// SIMATIC S7-200 SMART project (STEP 7-Micro/WIN SMART), CPU ST20

SYMBOL_TABLE System Symbols
Always_On        SM0.0    // Always ON
END_SYMBOL_TABLE

ORGANIZATION_BLOCK MAIN:OB1
TITLE=Program Comments
BEGIN
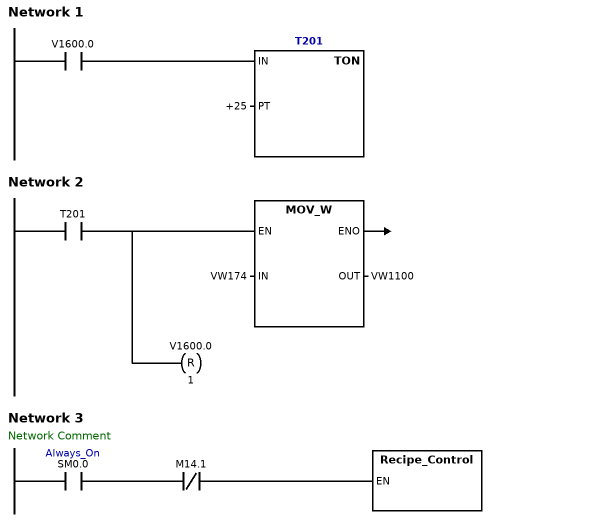
Network 1
LD     V1600.0
TON    T201, +25
Network 2
LD     T201
MOVW   VW174, VW1100
R      V1600.0, 1
Network 3
// Network Comment
LD     Always_On:SM0.0
AN     M14.1
CALL   Recipe_Control:SBR0
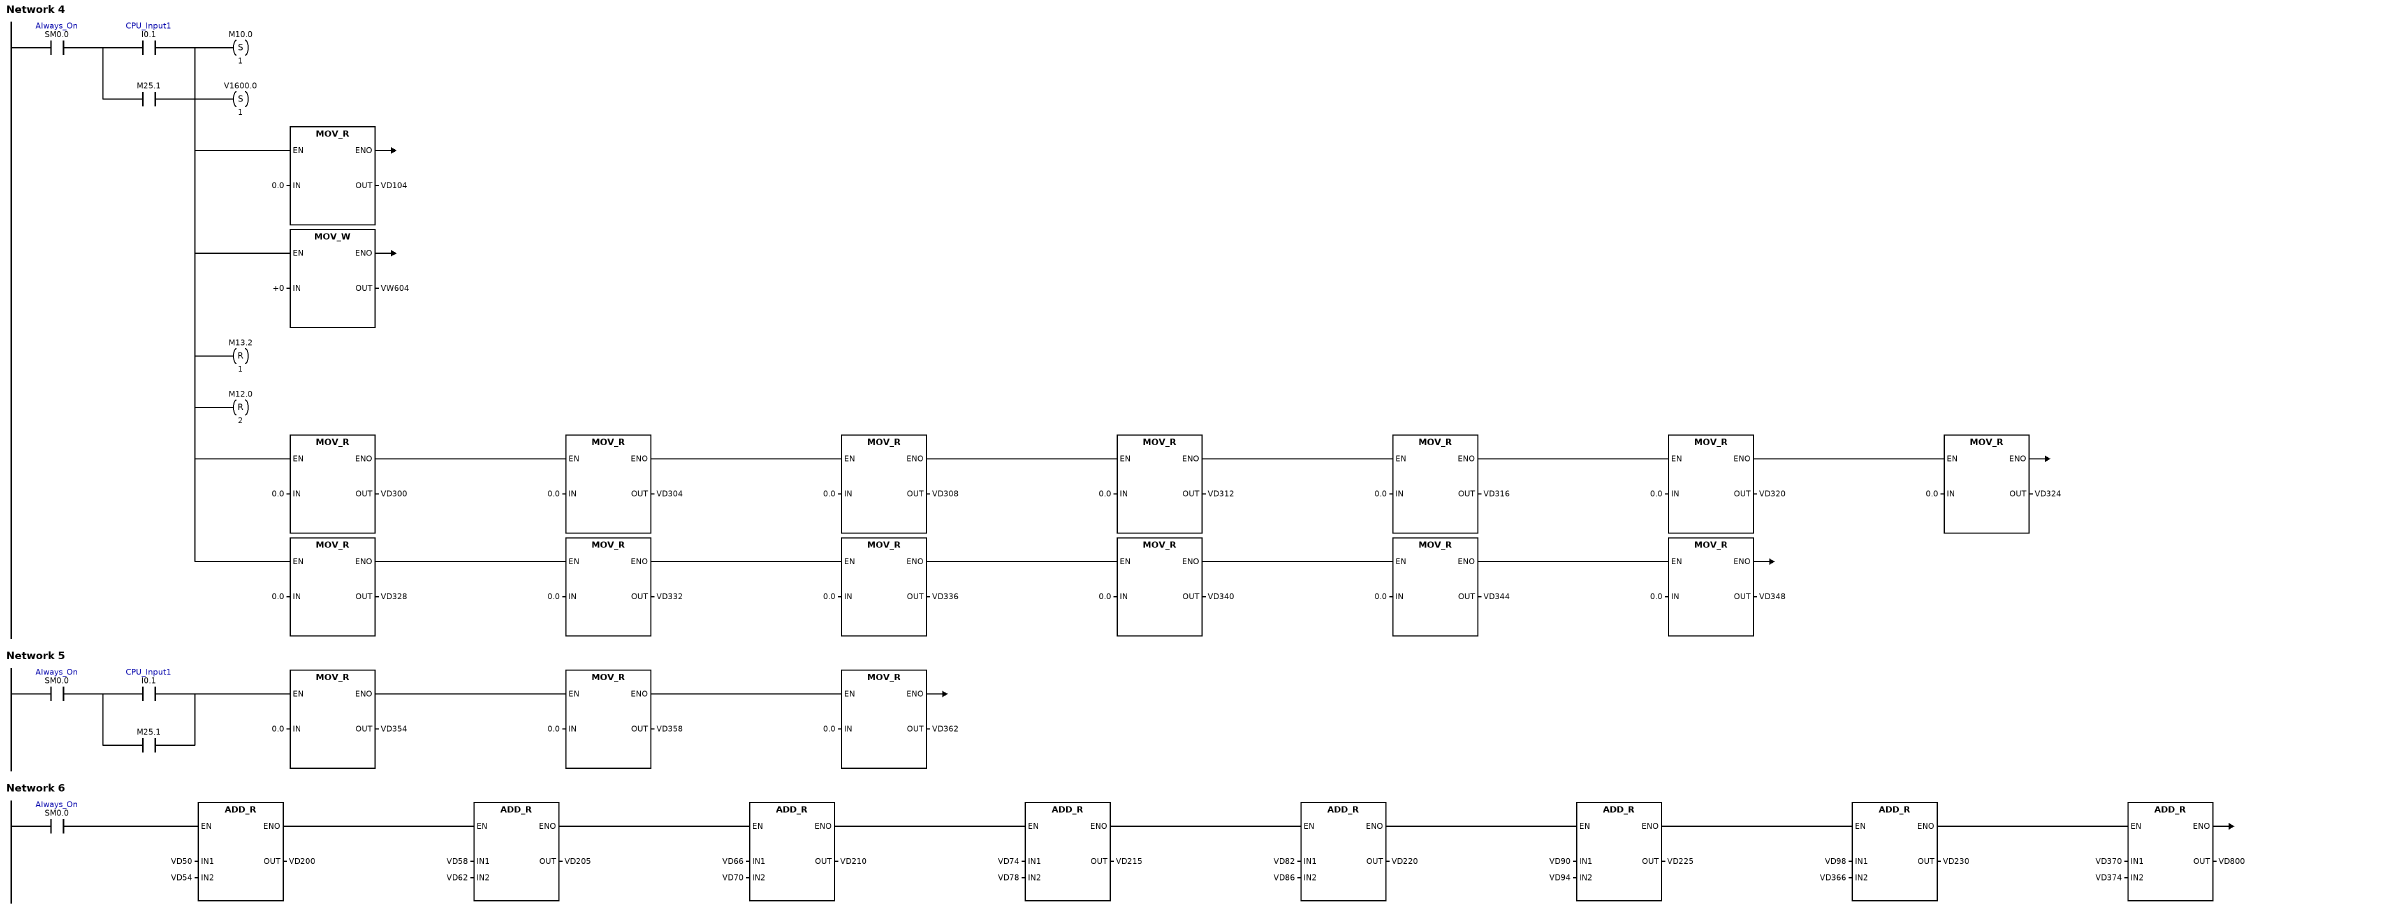
Network 4
LD     Always_On:SM0.0
LD     CPU_Input1:I0.1
O      M25.1
ALD
LPS
S      M10.0, 1
S      V1600.0, 1
MOVR   0.0, VD104
MOVW   +0, VW604
R      M13.2, 1
R      M12.0, 2
MOVR   0.0, VD300
AENO
MOVR   0.0, VD304
AENO
MOVR   0.0, VD308
AENO
MOVR   0.0, VD312
AENO
MOVR   0.0, VD316
AENO
MOVR   0.0, VD320
AENO
MOVR   0.0, VD324
LPP
MOVR   0.0, VD328
AENO
MOVR   0.0, VD332
AENO
MOVR   0.0, VD336
AENO
MOVR   0.0, VD340
AENO
MOVR   0.0, VD344
AENO
MOVR   0.0, VD348
Network 5
LD     Always_On:SM0.0
LD     CPU_Input1:I0.1
O      M25.1
ALD
MOVR   0.0, VD354
AENO
MOVR   0.0, VD358
AENO
MOVR   0.0, VD362
Network 6
LD     Always_On:SM0.0
MOVR   VD50, VD200
AENO
+R     VD54, VD200
AENO
MOVR   VD58, VD205
AENO
+R     VD62, VD205
AENO
MOVR   VD66, VD210
AENO
+R     VD70, VD210
AENO
MOVR   VD74, VD215
AENO
+R     VD78, VD215
AENO
MOVR   VD82, VD220
AENO
+R     VD86, VD220
AENO
MOVR   VD90, VD225
AENO
+R     VD94, VD225
AENO
MOVR   VD98, VD230
AENO
+R     VD366, VD230
AENO
MOVR   VD370, VD800
+R     VD374, VD800
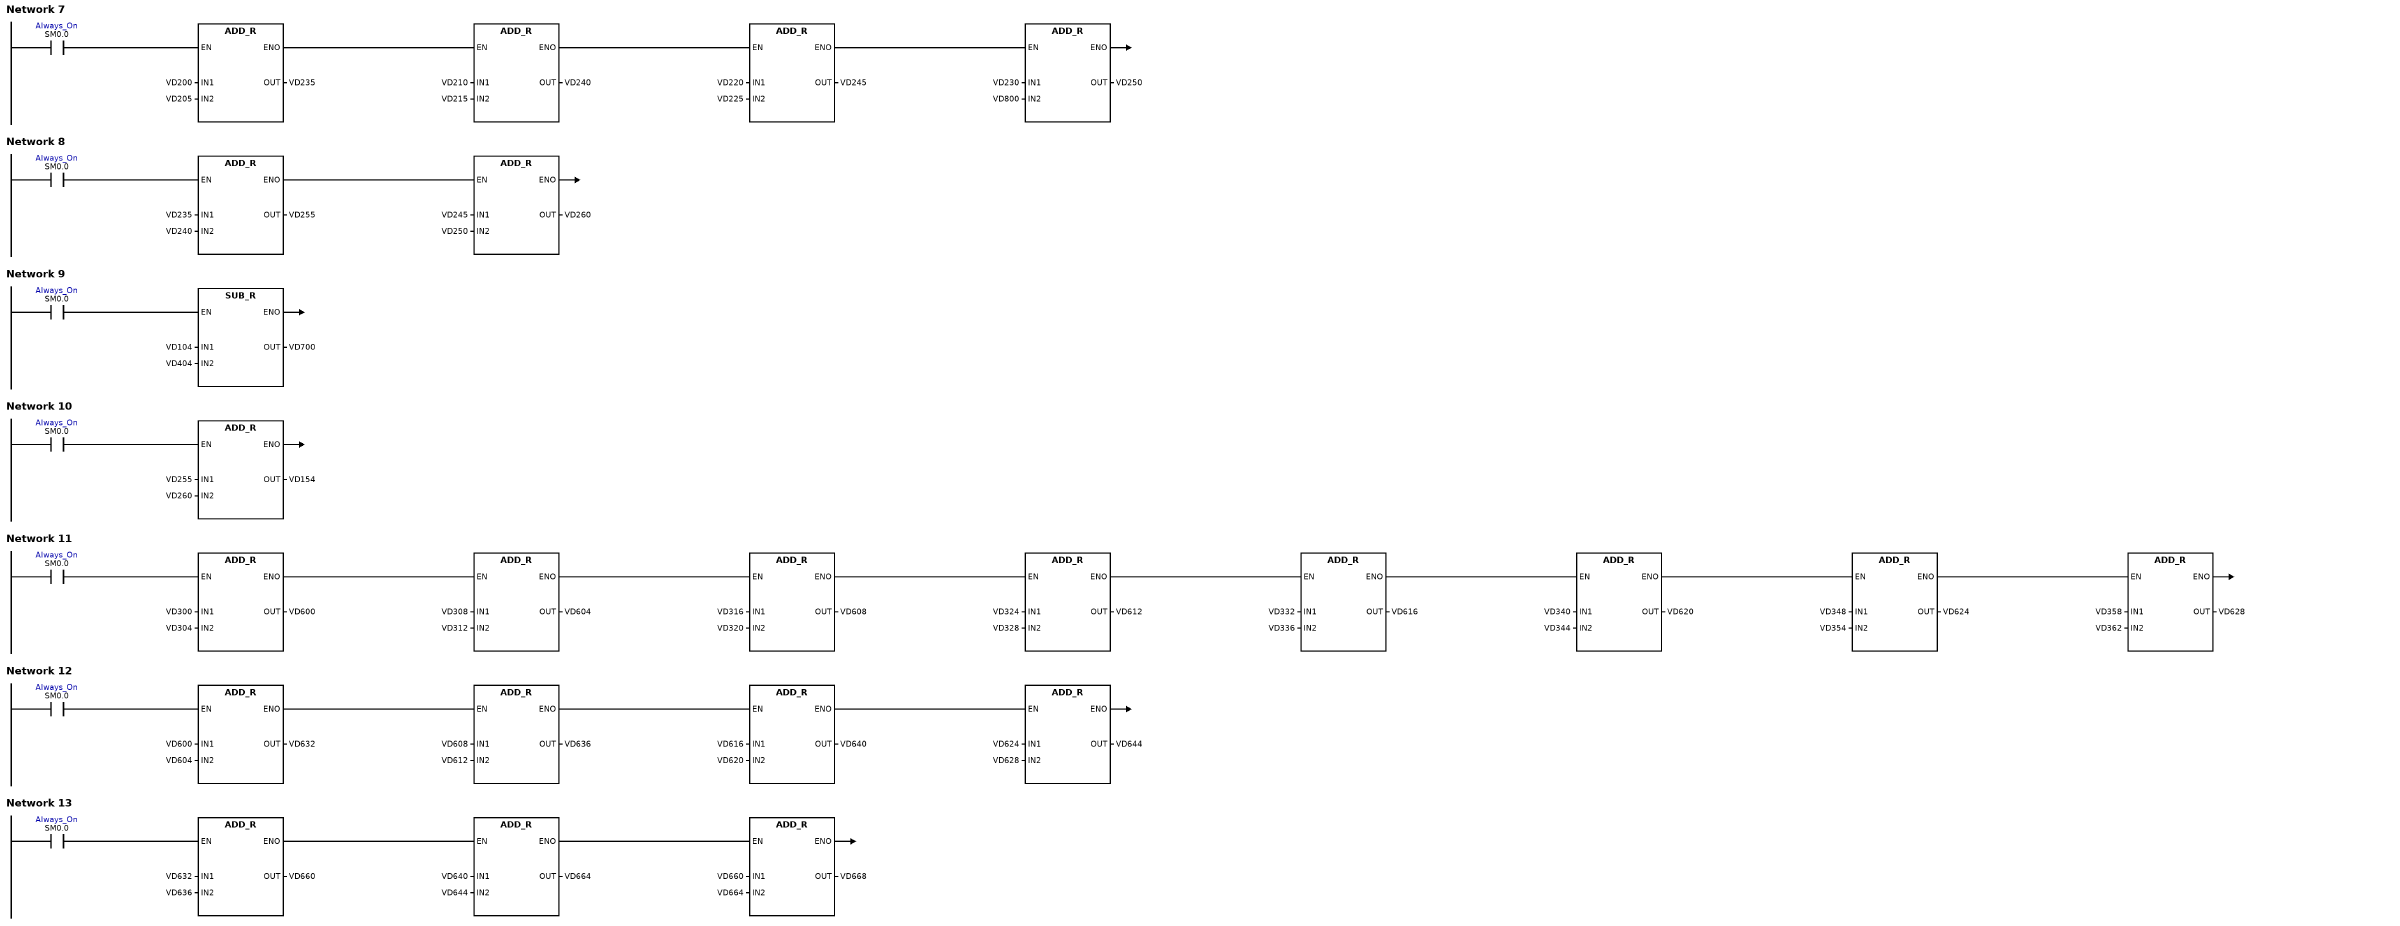
Network 7
LD     Always_On:SM0.0
MOVR   VD200, VD235
AENO
+R     VD205, VD235
AENO
MOVR   VD210, VD240
AENO
+R     VD215, VD240
AENO
MOVR   VD220, VD245
AENO
+R     VD225, VD245
AENO
MOVR   VD230, VD250
+R     VD800, VD250
Network 8
LD     Always_On:SM0.0
MOVR   VD235, VD255
AENO
+R     VD240, VD255
AENO
MOVR   VD245, VD260
+R     VD250, VD260
Network 9
LD     Always_On:SM0.0
MOVR   VD104, VD700
-R     VD404, VD700
Network 10
LD     Always_On:SM0.0
MOVR   VD255, VD154
+R     VD260, VD154
Network 11
LD     Always_On:SM0.0
MOVR   VD300, VD600
AENO
+R     VD304, VD600
AENO
MOVR   VD308, VD604
AENO
+R     VD312, VD604
AENO
MOVR   VD316, VD608
AENO
+R     VD320, VD608
AENO
MOVR   VD324, VD612
AENO
+R     VD328, VD612
AENO
MOVR   VD332, VD616
AENO
+R     VD336, VD616
AENO
MOVR   VD340, VD620
AENO
+R     VD344, VD620
AENO
MOVR   VD348, VD624
AENO
+R     VD354, VD624
AENO
MOVR   VD358, VD628
+R     VD362, VD628
Network 12
LD     Always_On:SM0.0
MOVR   VD600, VD632
AENO
+R     VD604, VD632
AENO
MOVR   VD608, VD636
AENO
+R     VD612, VD636
AENO
MOVR   VD616, VD640
AENO
+R     VD620, VD640
AENO
MOVR   VD624, VD644
+R     VD628, VD644
Network 13
LD     Always_On:SM0.0
MOVR   VD632, VD660
AENO
+R     VD636, VD660
AENO
MOVR   VD640, VD664
AENO
+R     VD644, VD664
AENO
MOVR   VD660, VD668
+R     VD664, VD668
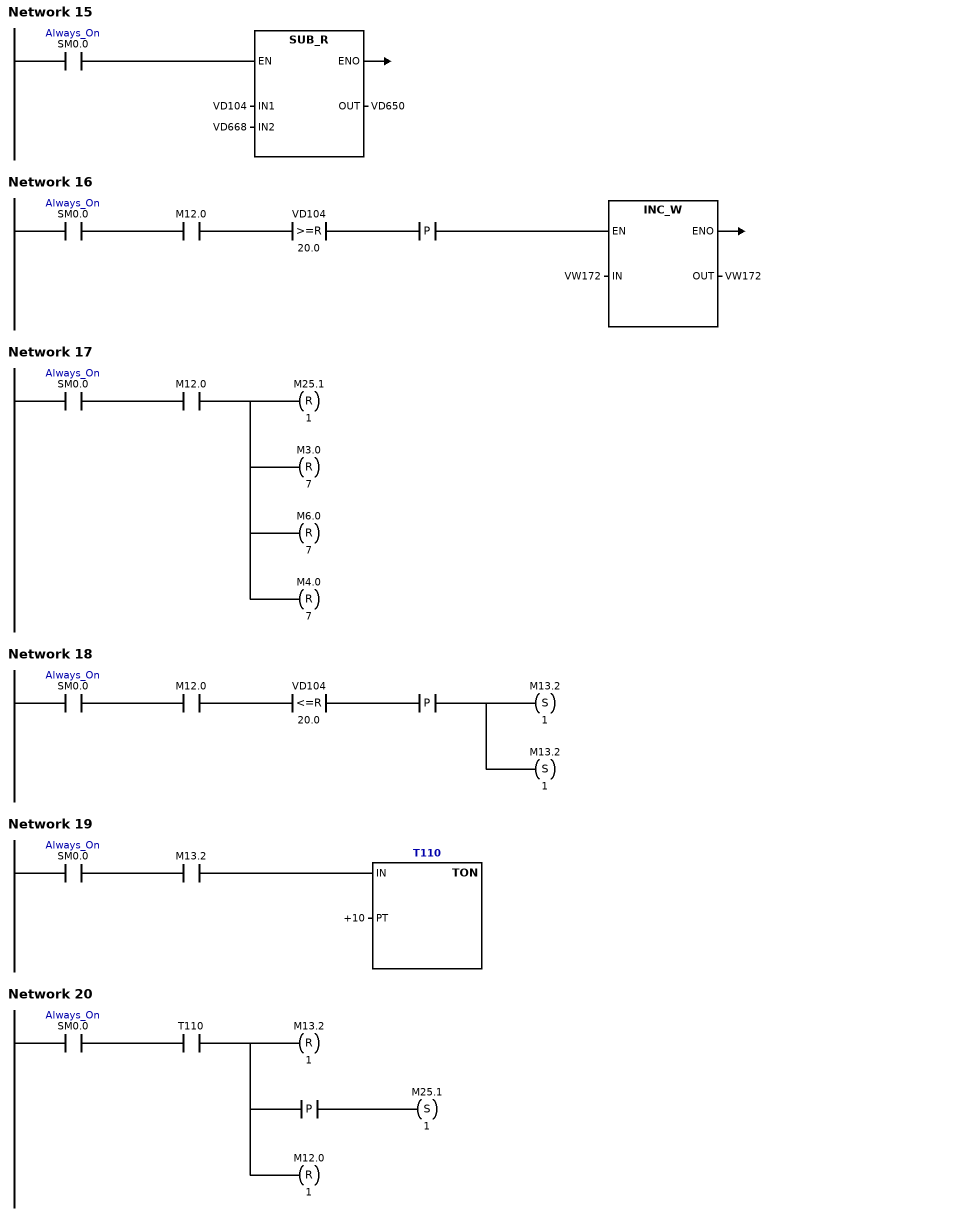
Network 15
LD     Always_On:SM0.0
MOVR   VD104, VD650
-R     VD668, VD650
Network 16
LD     Always_On:SM0.0
A      M12.0
AR>=   VD104, 20.0
EU
INCW   VW172
Network 17
LD     Always_On:SM0.0
A      M12.0
R      M25.1, 1
R      M3.0, 7
R      M6.0, 7
R      M4.0, 7
Network 18
LD     Always_On:SM0.0
A      M12.0
AR<=   VD104, 20.0
EU
S      M13.2, 1
S      M13.2, 1
Network 19
LD     Always_On:SM0.0
A      M13.2
TON    T110, +10
Network 20
LD     Always_On:SM0.0
A      T110
LPS
R      M13.2, 1
EU
S      M25.1, 1
LPP
R      M12.0, 1
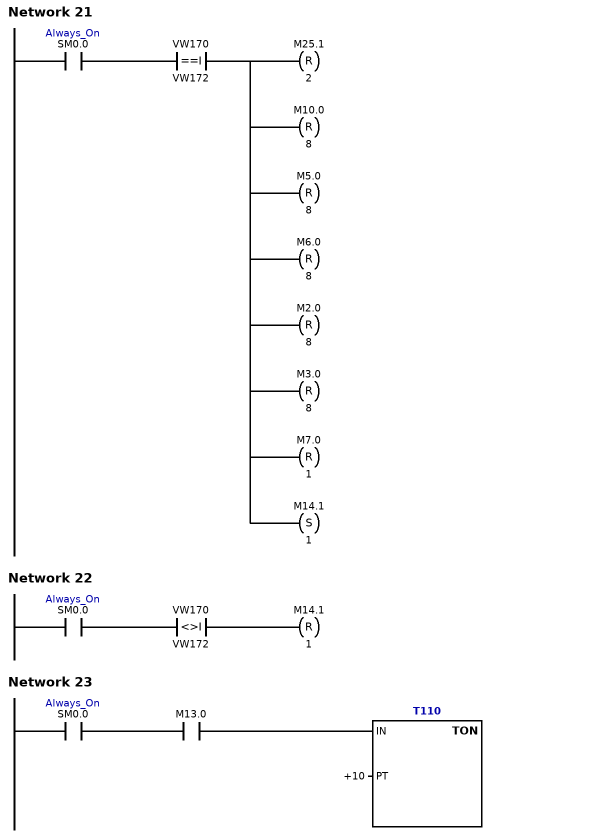
Network 21
LD     Always_On:SM0.0
AW=    VW170, VW172
R      M25.1, 2
R      M10.0, 8
R      M5.0, 8
R      M6.0, 8
R      M2.0, 8
R      M3.0, 8
R      M7.0, 1
S      M14.1, 1
Network 22
LD     Always_On:SM0.0
AW<>   VW170, VW172
R      M14.1, 1
Network 23
LD     Always_On:SM0.0
A      M13.0
TON    T110, +10
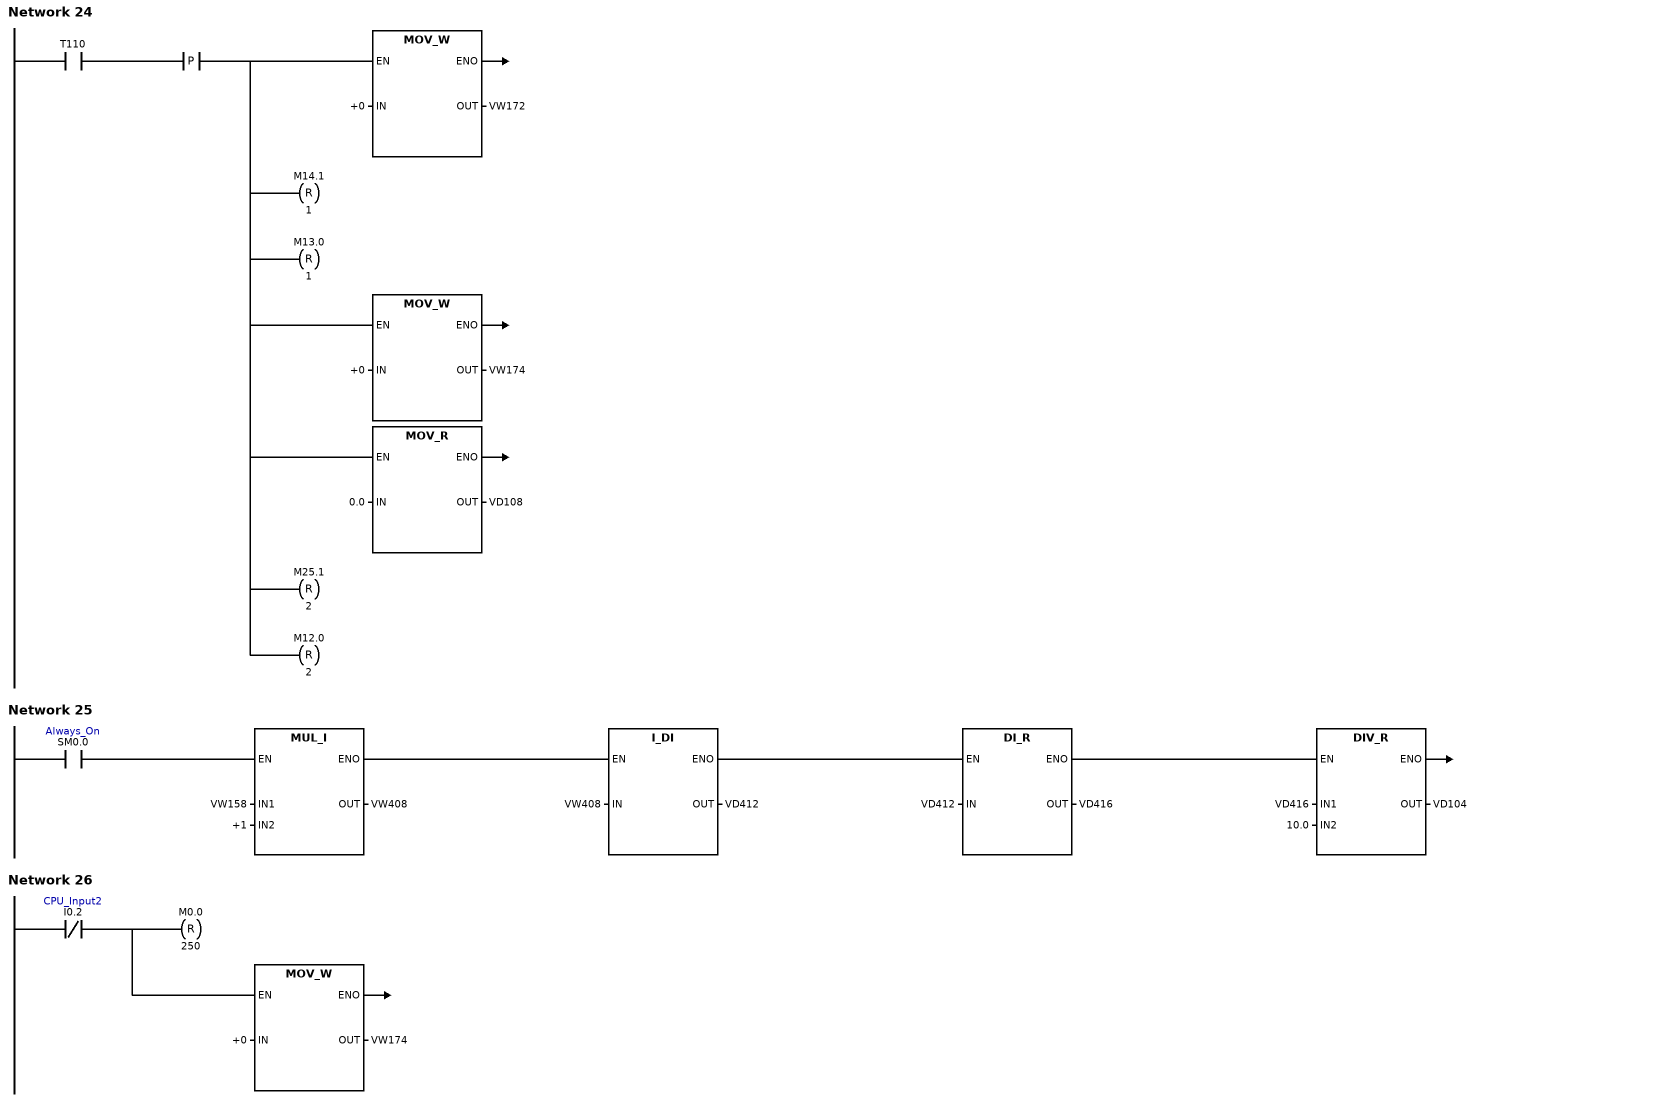
Network 24
LD     T110
EU
MOVW   +0, VW172
R      M14.1, 1
R      M13.0, 1
MOVW   +0, VW174
MOVR   0.0, VD108
R      M25.1, 2
R      M12.0, 2
Network 25
LD     Always_On:SM0.0
MOVW   VW158, VW408
AENO
*I     +1, VW408
AENO
ITD    VW408, VD412
AENO
DTR    VD412, VD416
AENO
MOVR   VD416, VD104
/R     10.0, VD104
Network 26
LDN    CPU_Input2:I0.2
R      M0.0, 250
MOVW   +0, VW174
END_ORGANIZATION_BLOCK

SUBROUTINE_BLOCK Recipe_Control:SBR0
TITLE=Subroutine Comments
BEGIN
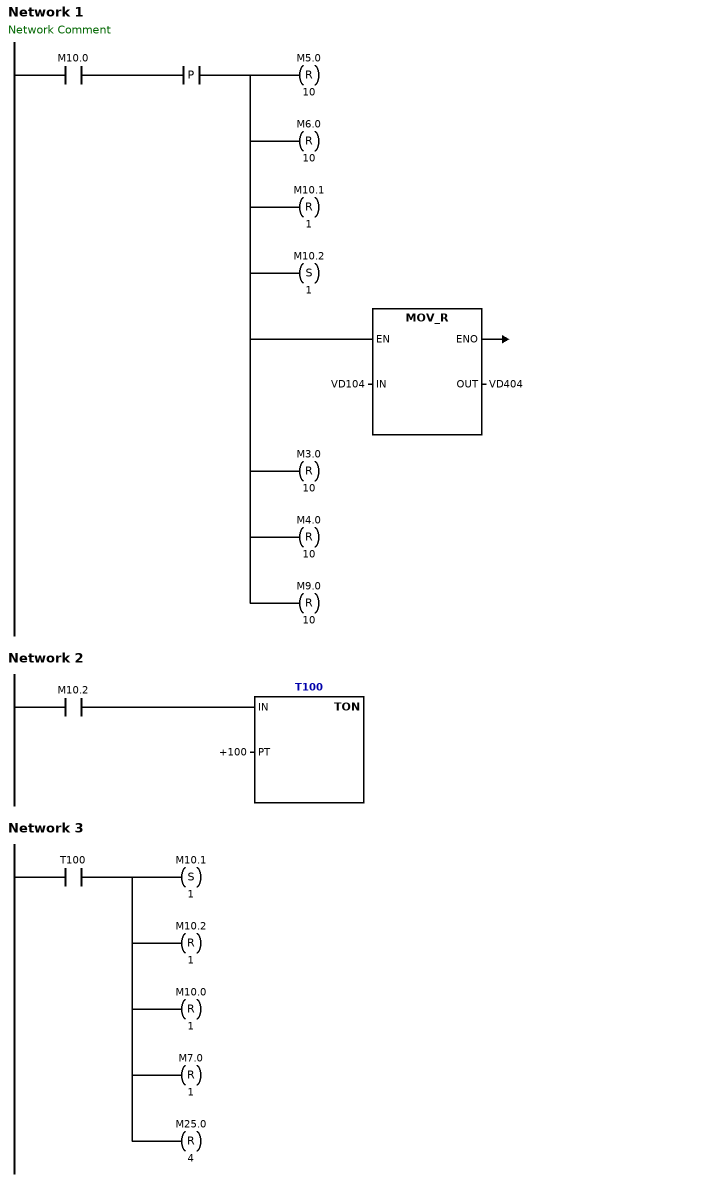
Network 1
// Network Comment
LD     M10.0
EU
R      M5.0, 10
R      M6.0, 10
R      M10.1, 1
S      M10.2, 1
MOVR   VD104, VD404
R      M3.0, 10
R      M4.0, 10
R      M9.0, 10
Network 2
LD     M10.2
TON    T100, +100
Network 3
LD     T100
S      M10.1, 1
R      M10.2, 1
R      M10.0, 1
R      M7.0, 1
R      M25.0, 4
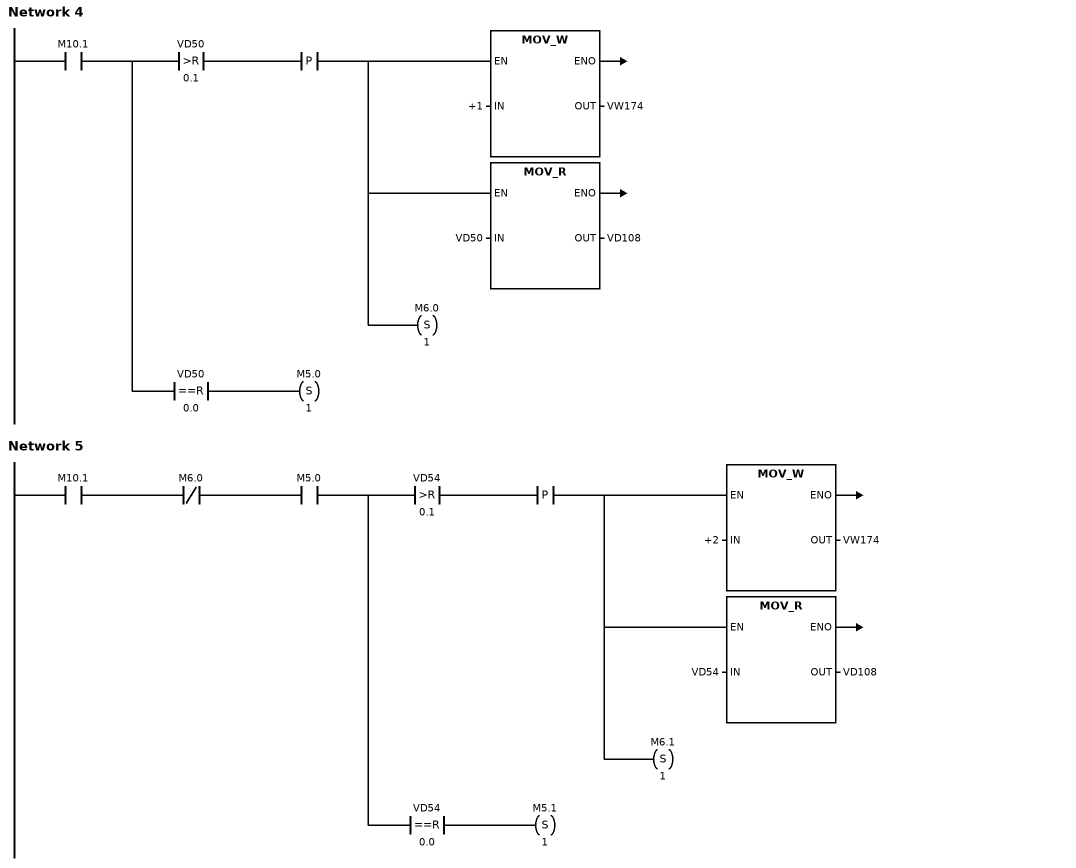
Network 4
LD     M10.1
LPS
AR>    VD50, 0.1
EU
MOVW   +1, VW174
MOVR   VD50, VD108
S      M6.0, 1
LPP
AR=    VD50, 0.0
S      M5.0, 1
Network 5
LD     M10.1
AN     M6.0
A      M5.0
LPS
AR>    VD54, 0.1
EU
MOVW   +2, VW174
MOVR   VD54, VD108
S      M6.1, 1
LPP
AR=    VD54, 0.0
S      M5.1, 1
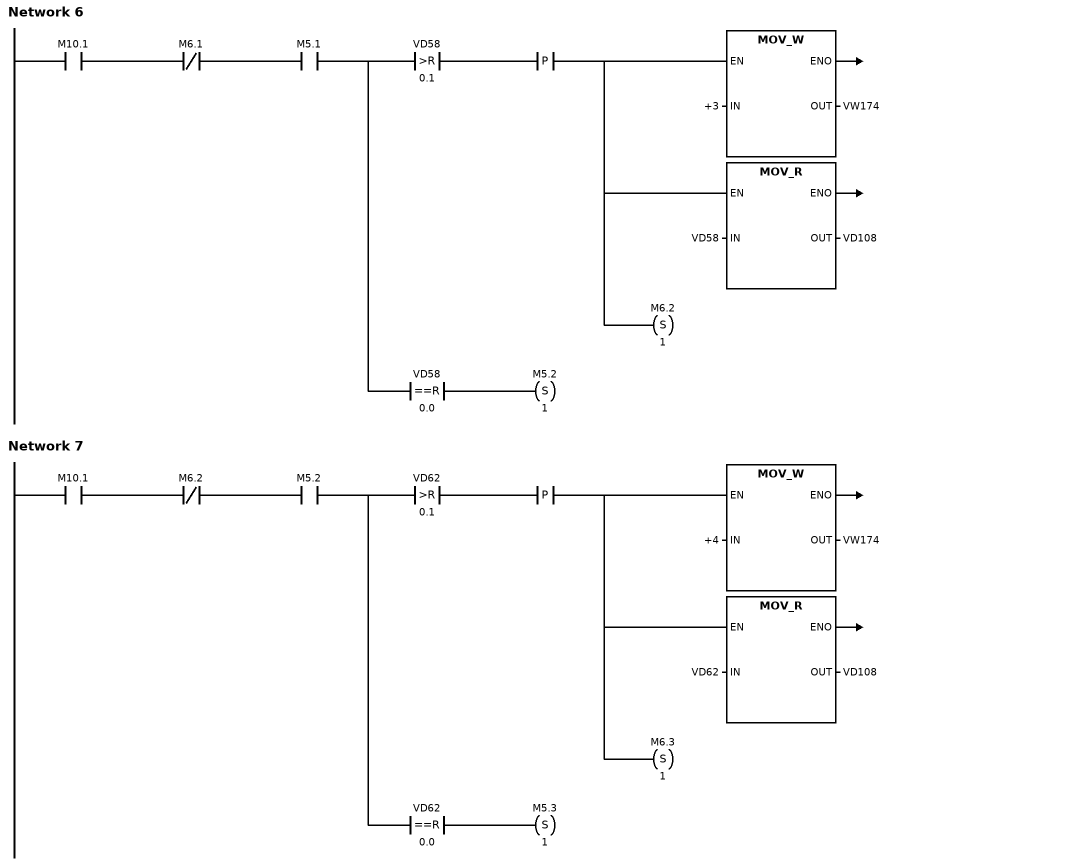
Network 6
LD     M10.1
AN     M6.1
A      M5.1
LPS
AR>    VD58, 0.1
EU
MOVW   +3, VW174
MOVR   VD58, VD108
S      M6.2, 1
LPP
AR=    VD58, 0.0
S      M5.2, 1
Network 7
LD     M10.1
AN     M6.2
A      M5.2
LPS
AR>    VD62, 0.1
EU
MOVW   +4, VW174
MOVR   VD62, VD108
S      M6.3, 1
LPP
AR=    VD62, 0.0
S      M5.3, 1
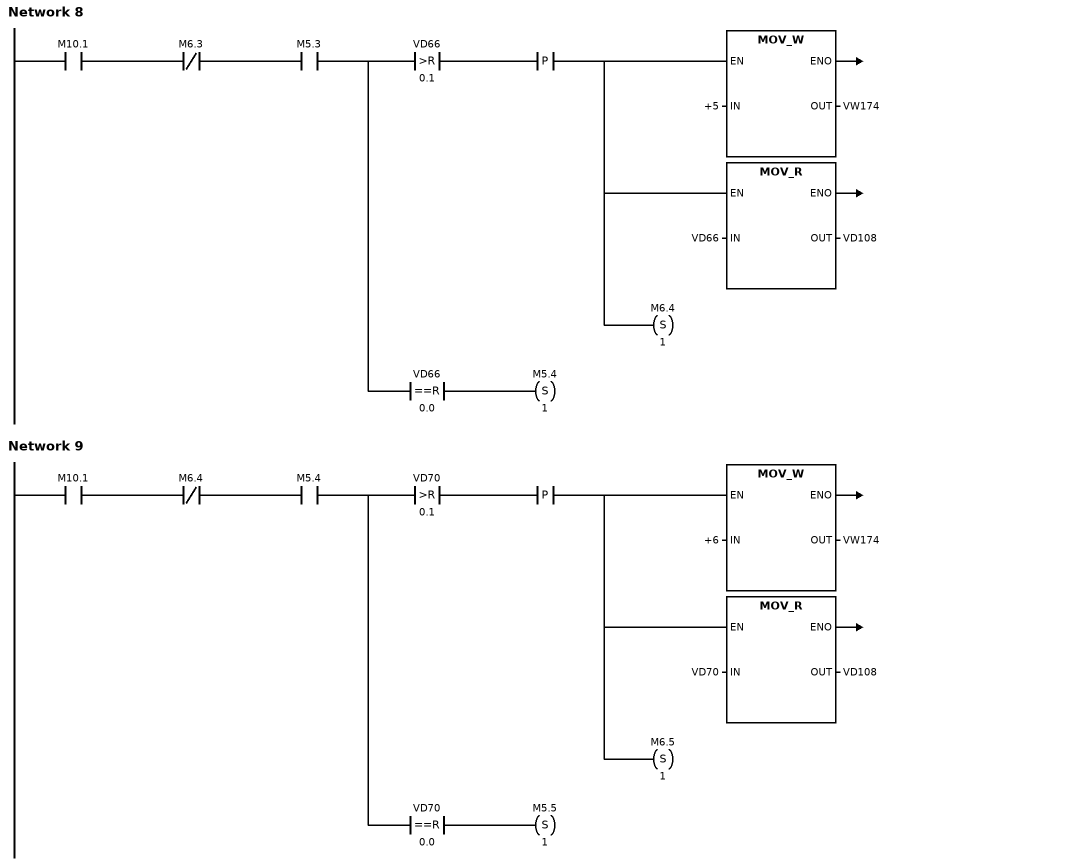
Network 8
LD     M10.1
AN     M6.3
A      M5.3
LPS
AR>    VD66, 0.1
EU
MOVW   +5, VW174
MOVR   VD66, VD108
S      M6.4, 1
LPP
AR=    VD66, 0.0
S      M5.4, 1
Network 9
LD     M10.1
AN     M6.4
A      M5.4
LPS
AR>    VD70, 0.1
EU
MOVW   +6, VW174
MOVR   VD70, VD108
S      M6.5, 1
LPP
AR=    VD70, 0.0
S      M5.5, 1
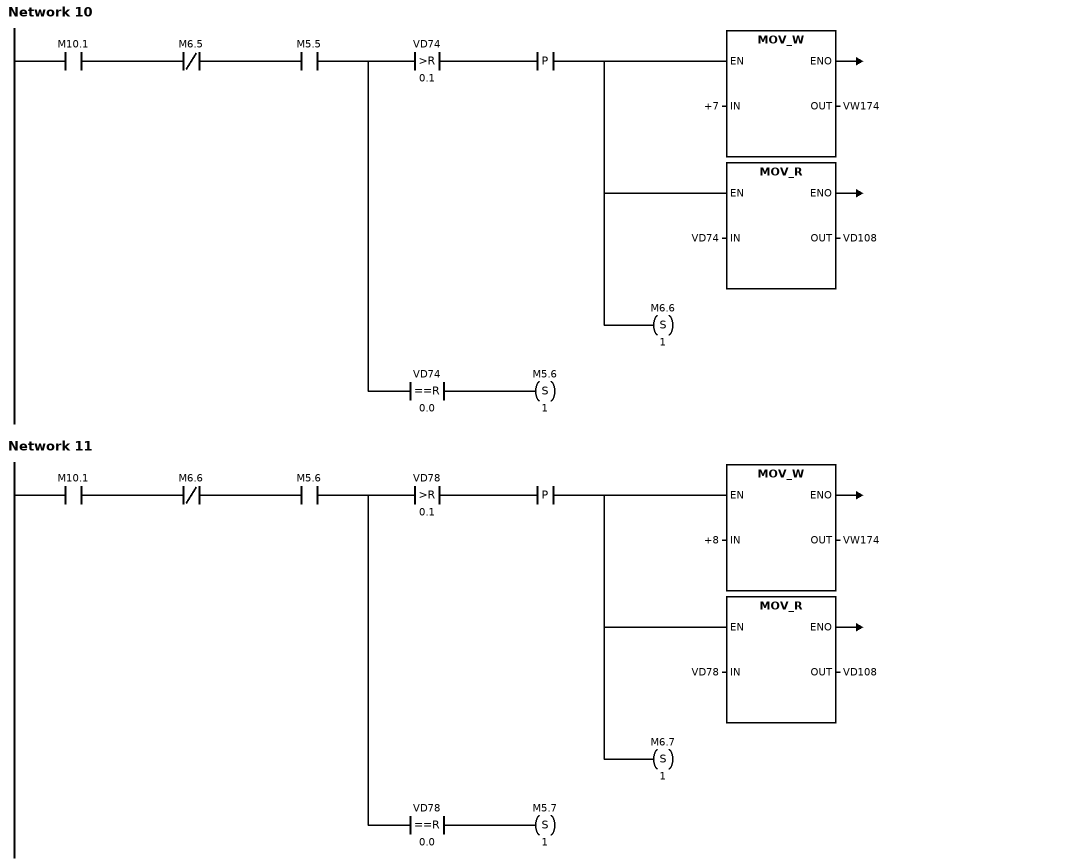
Network 10
LD     M10.1
AN     M6.5
A      M5.5
LPS
AR>    VD74, 0.1
EU
MOVW   +7, VW174
MOVR   VD74, VD108
S      M6.6, 1
LPP
AR=    VD74, 0.0
S      M5.6, 1
Network 11
LD     M10.1
AN     M6.6
A      M5.6
LPS
AR>    VD78, 0.1
EU
MOVW   +8, VW174
MOVR   VD78, VD108
S      M6.7, 1
LPP
AR=    VD78, 0.0
S      M5.7, 1
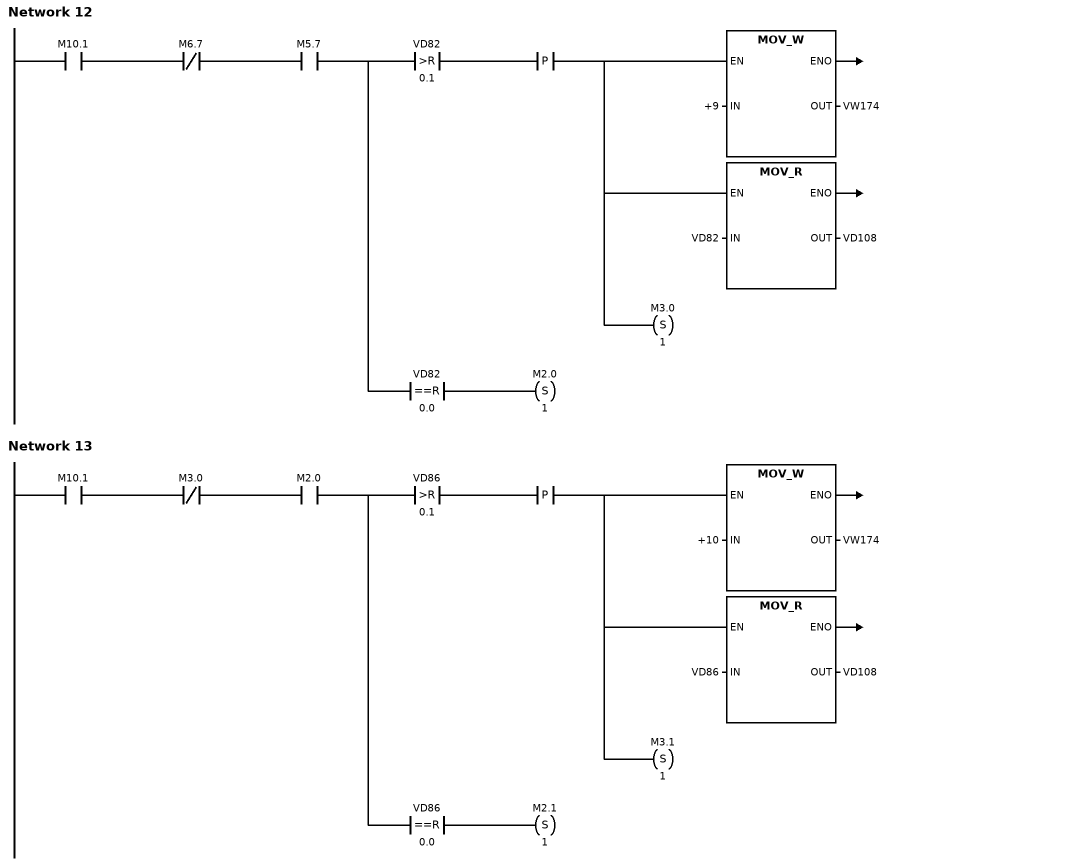
Network 12
LD     M10.1
AN     M6.7
A      M5.7
LPS
AR>    VD82, 0.1
EU
MOVW   +9, VW174
MOVR   VD82, VD108
S      M3.0, 1
LPP
AR=    VD82, 0.0
S      M2.0, 1
Network 13
LD     M10.1
AN     M3.0
A      M2.0
LPS
AR>    VD86, 0.1
EU
MOVW   +10, VW174
MOVR   VD86, VD108
S      M3.1, 1
LPP
AR=    VD86, 0.0
S      M2.1, 1
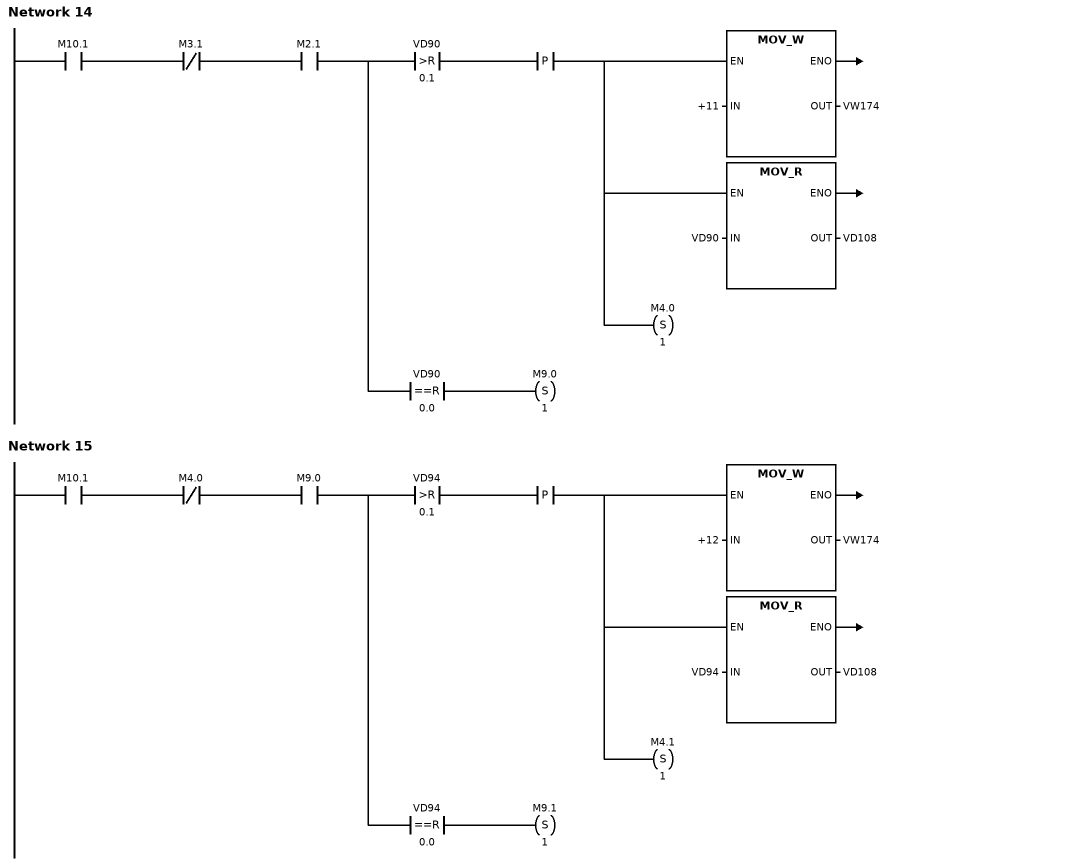
Network 14
LD     M10.1
AN     M3.1
A      M2.1
LPS
AR>    VD90, 0.1
EU
MOVW   +11, VW174
MOVR   VD90, VD108
S      M4.0, 1
LPP
AR=    VD90, 0.0
S      M9.0, 1
Network 15
LD     M10.1
AN     M4.0
A      M9.0
LPS
AR>    VD94, 0.1
EU
MOVW   +12, VW174
MOVR   VD94, VD108
S      M4.1, 1
LPP
AR=    VD94, 0.0
S      M9.1, 1
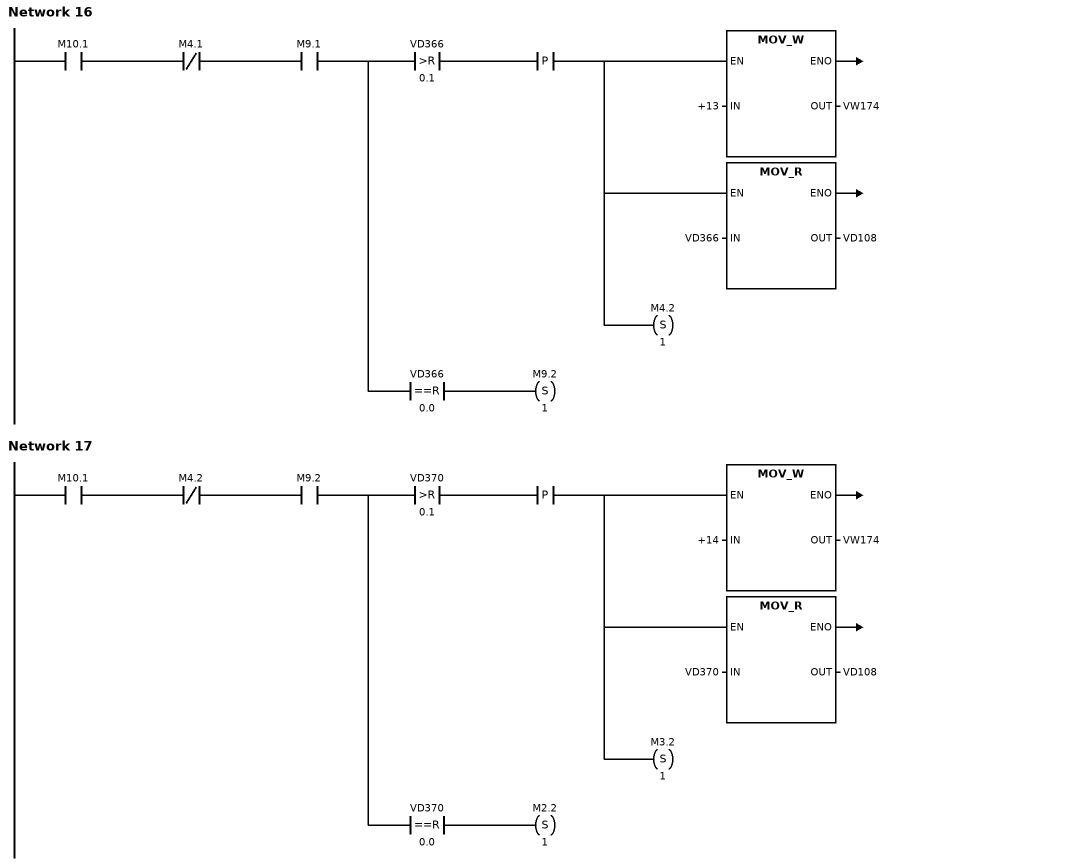
Network 16
LD     M10.1
AN     M4.1
A      M9.1
LPS
AR>    VD366, 0.1
EU
MOVW   +13, VW174
MOVR   VD366, VD108
S      M4.2, 1
LPP
AR=    VD366, 0.0
S      M9.2, 1
Network 17
LD     M10.1
AN     M4.2
A      M9.2
LPS
AR>    VD370, 0.1
EU
MOVW   +14, VW174
MOVR   VD370, VD108
S      M3.2, 1
LPP
AR=    VD370, 0.0
S      M2.2, 1
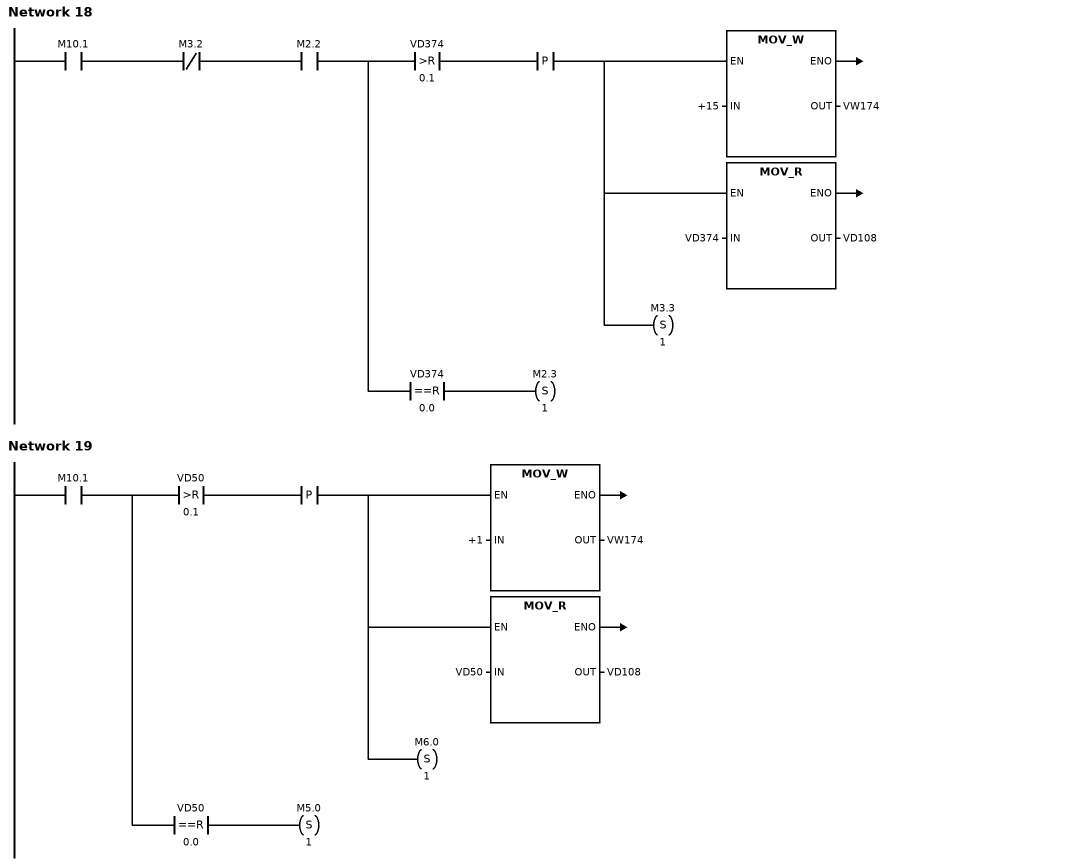
Network 18
LD     M10.1
AN     M3.2
A      M2.2
LPS
AR>    VD374, 0.1
EU
MOVW   +15, VW174
MOVR   VD374, VD108
S      M3.3, 1
LPP
AR=    VD374, 0.0
S      M2.3, 1
Network 19
LD     M10.1
LPS
AR>    VD50, 0.1
EU
MOVW   +1, VW174
MOVR   VD50, VD108
S      M6.0, 1
LPP
AR=    VD50, 0.0
S      M5.0, 1
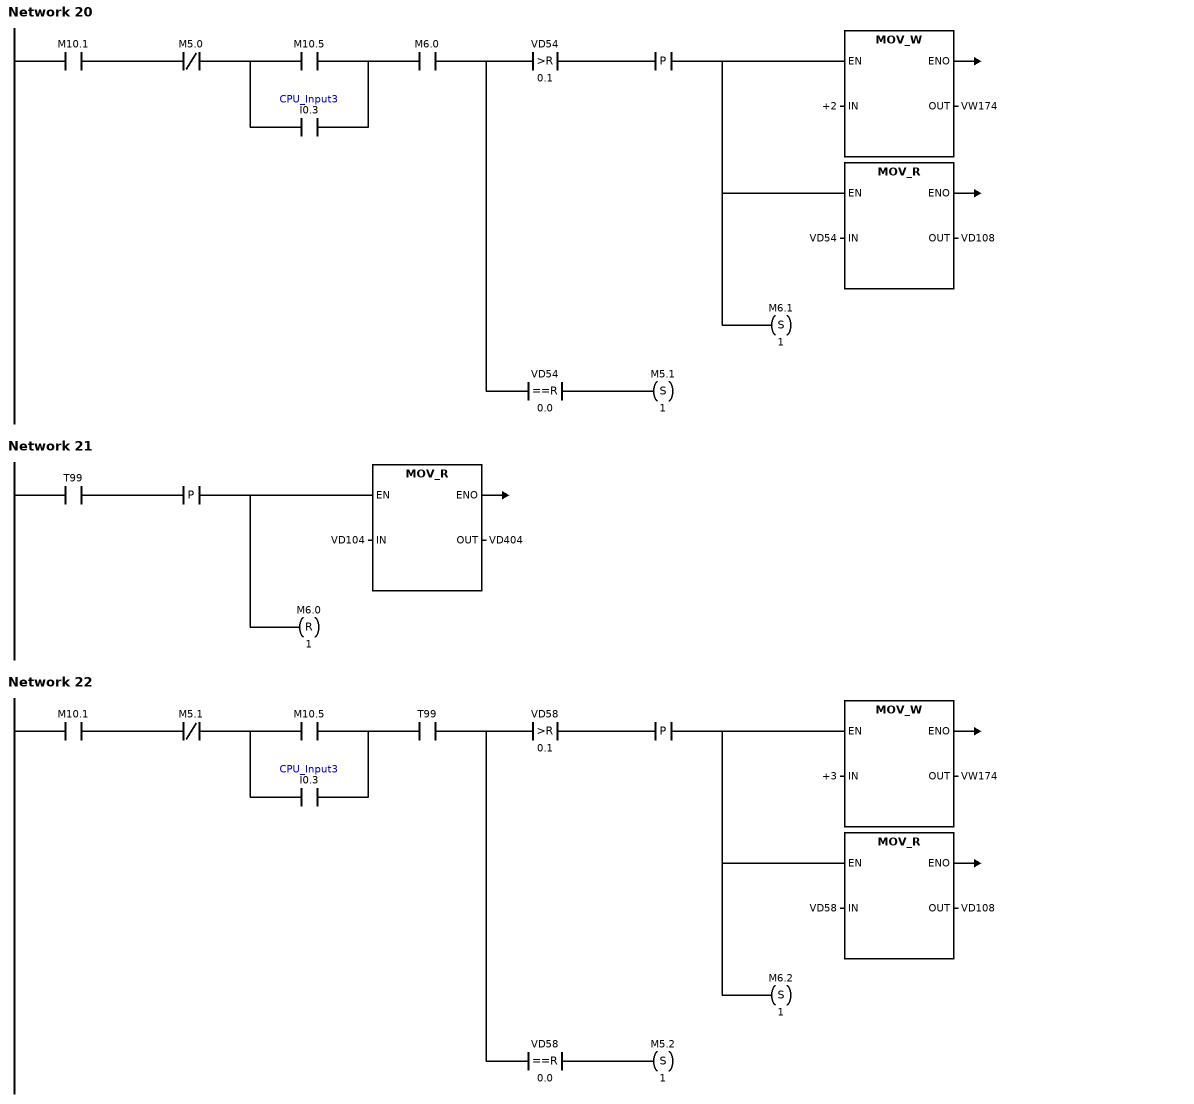
Network 20
LD     M10.1
AN     M5.0
LD     M10.5
O      CPU_Input3:I0.3
ALD
A      M6.0
LPS
AR>    VD54, 0.1
EU
MOVW   +2, VW174
MOVR   VD54, VD108
S      M6.1, 1
LPP
AR=    VD54, 0.0
S      M5.1, 1
Network 21
LD     T99
EU
MOVR   VD104, VD404
R      M6.0, 1
Network 22
LD     M10.1
AN     M5.1
LD     M10.5
O      CPU_Input3:I0.3
ALD
A      T99
LPS
AR>    VD58, 0.1
EU
MOVW   +3, VW174
MOVR   VD58, VD108
S      M6.2, 1
LPP
AR=    VD58, 0.0
S      M5.2, 1
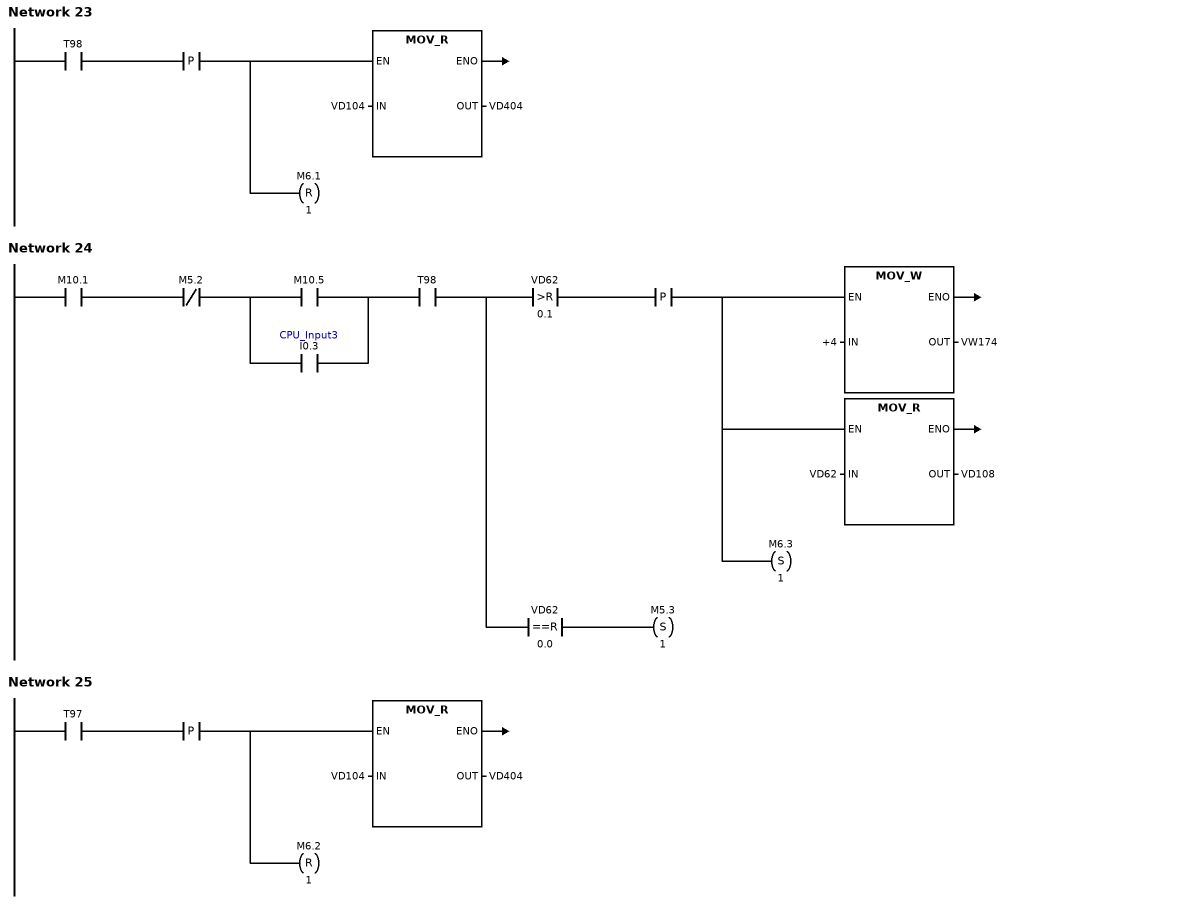
Network 23
LD     T98
EU
MOVR   VD104, VD404
R      M6.1, 1
Network 24
LD     M10.1
AN     M5.2
LD     M10.5
O      CPU_Input3:I0.3
ALD
A      T98
LPS
AR>    VD62, 0.1
EU
MOVW   +4, VW174
MOVR   VD62, VD108
S      M6.3, 1
LPP
AR=    VD62, 0.0
S      M5.3, 1
Network 25
LD     T97
EU
MOVR   VD104, VD404
R      M6.2, 1
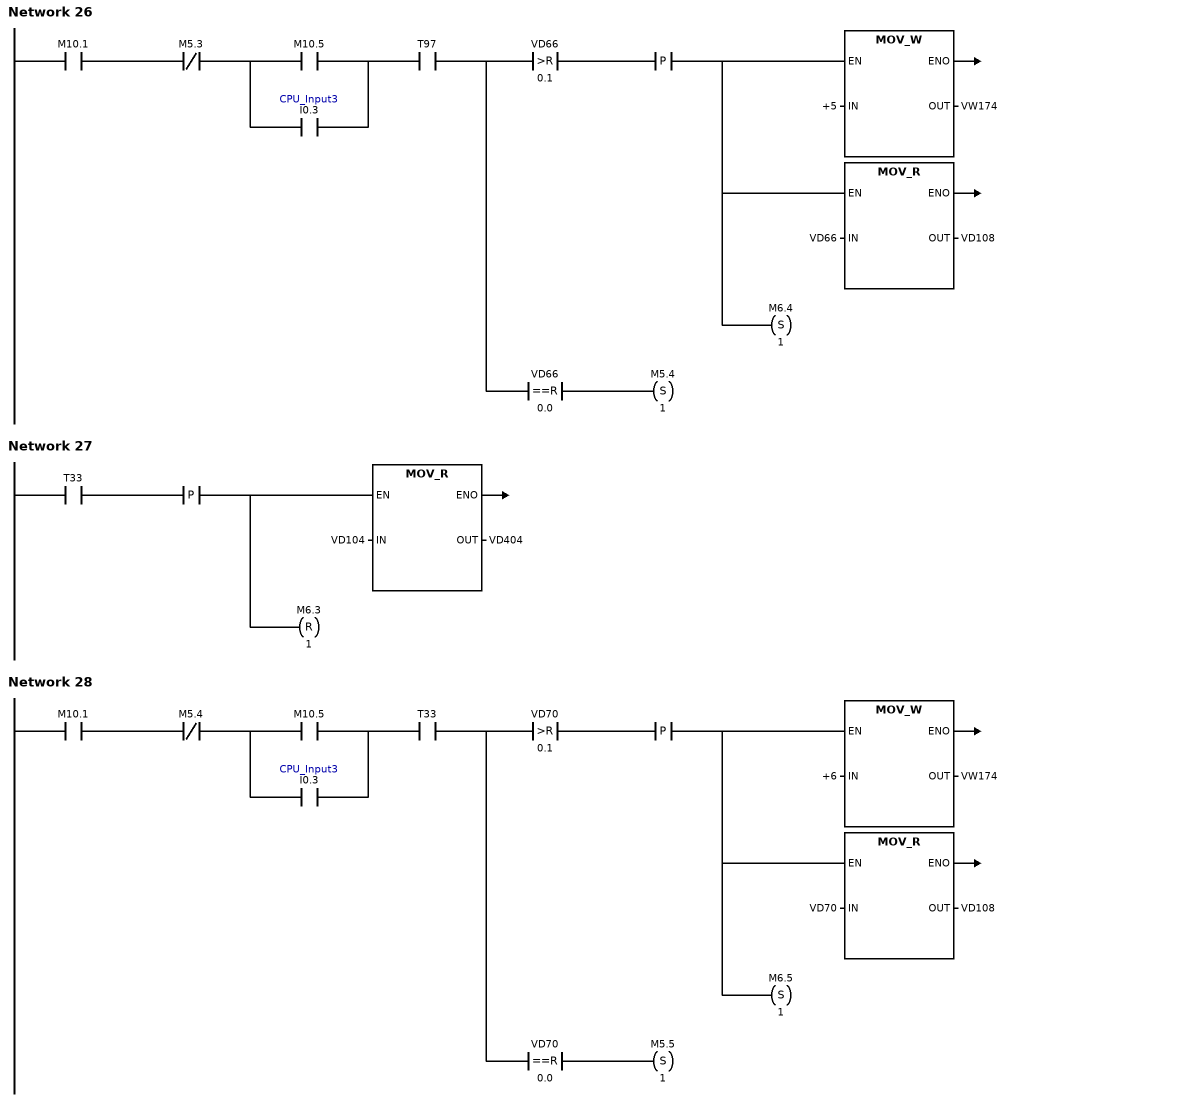
Network 26
LD     M10.1
AN     M5.3
LD     M10.5
O      CPU_Input3:I0.3
ALD
A      T97
LPS
AR>    VD66, 0.1
EU
MOVW   +5, VW174
MOVR   VD66, VD108
S      M6.4, 1
LPP
AR=    VD66, 0.0
S      M5.4, 1
Network 27
LD     T33
EU
MOVR   VD104, VD404
R      M6.3, 1
Network 28
LD     M10.1
AN     M5.4
LD     M10.5
O      CPU_Input3:I0.3
ALD
A      T33
LPS
AR>    VD70, 0.1
EU
MOVW   +6, VW174
MOVR   VD70, VD108
S      M6.5, 1
LPP
AR=    VD70, 0.0
S      M5.5, 1
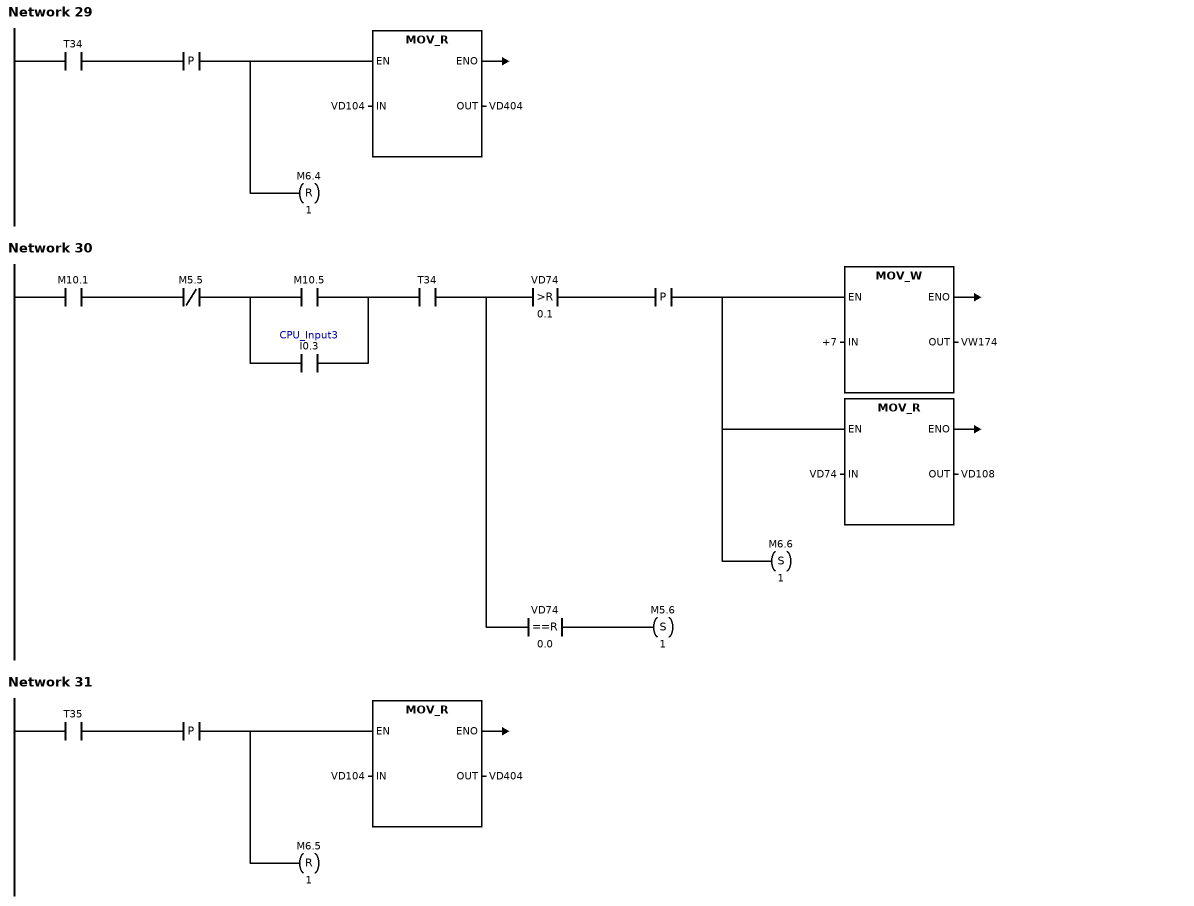
Network 29
LD     T34
EU
MOVR   VD104, VD404
R      M6.4, 1
Network 30
LD     M10.1
AN     M5.5
LD     M10.5
O      CPU_Input3:I0.3
ALD
A      T34
LPS
AR>    VD74, 0.1
EU
MOVW   +7, VW174
MOVR   VD74, VD108
S      M6.6, 1
LPP
AR=    VD74, 0.0
S      M5.6, 1
Network 31
LD     T35
EU
MOVR   VD104, VD404
R      M6.5, 1
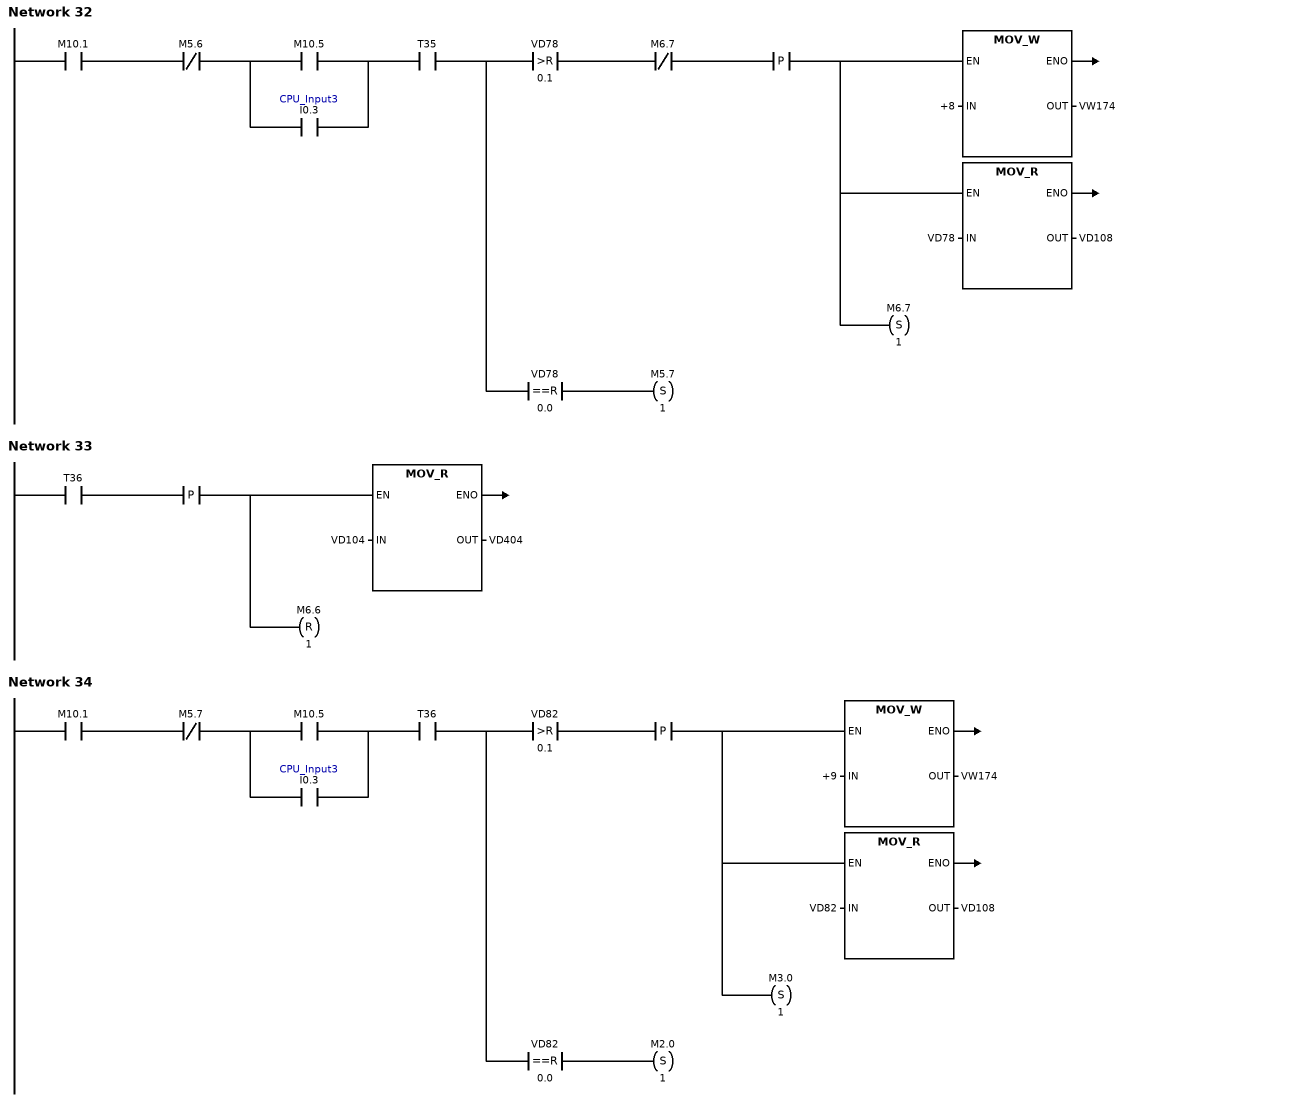
Network 32
LD     M10.1
AN     M5.6
LD     M10.5
O      CPU_Input3:I0.3
ALD
A      T35
LPS
AR>    VD78, 0.1
AN     M6.7
EU
MOVW   +8, VW174
MOVR   VD78, VD108
S      M6.7, 1
LPP
AR=    VD78, 0.0
S      M5.7, 1
Network 33
LD     T36
EU
MOVR   VD104, VD404
R      M6.6, 1
Network 34
LD     M10.1
AN     M5.7
LD     M10.5
O      CPU_Input3:I0.3
ALD
A      T36
LPS
AR>    VD82, 0.1
EU
MOVW   +9, VW174
MOVR   VD82, VD108
S      M3.0, 1
LPP
AR=    VD82, 0.0
S      M2.0, 1
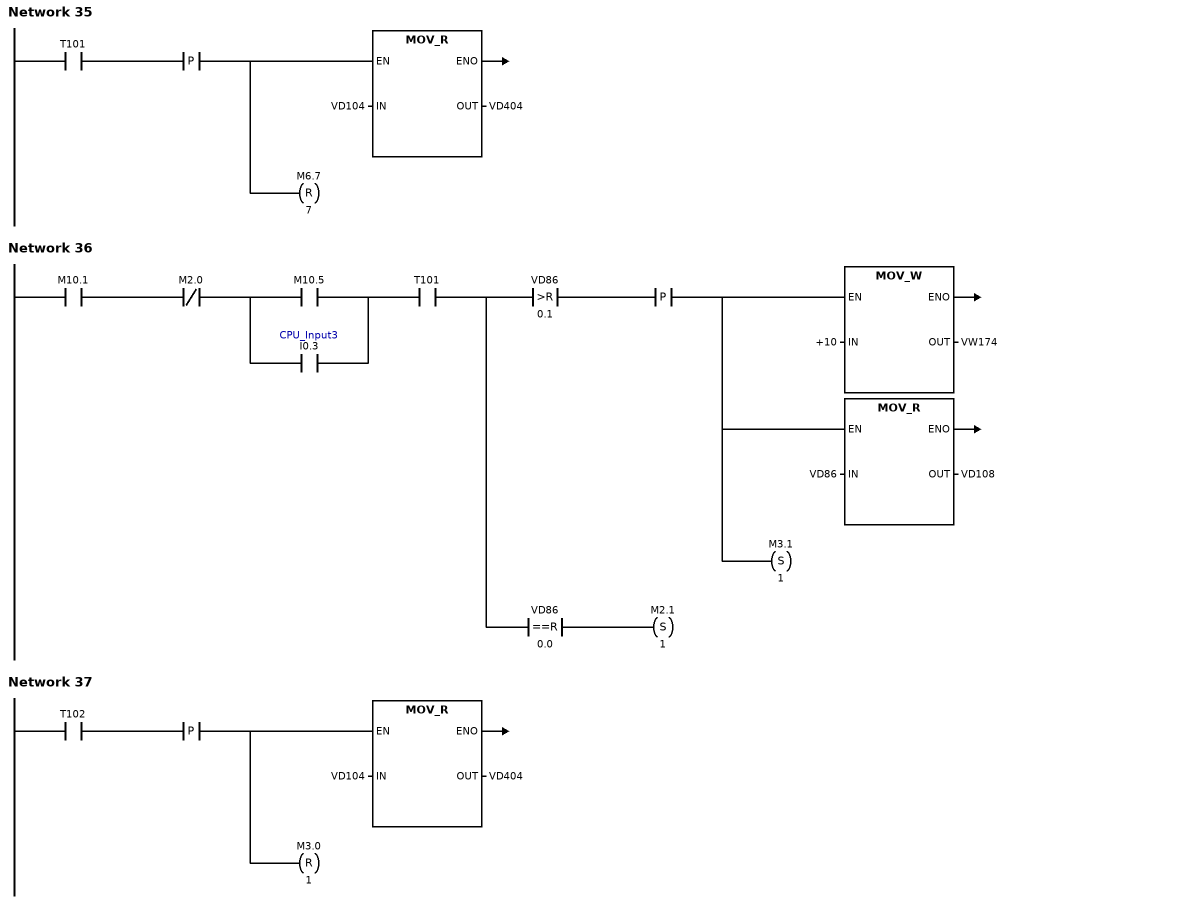
Network 35
LD     T101
EU
MOVR   VD104, VD404
R      M6.7, 7
Network 36
LD     M10.1
AN     M2.0
LD     M10.5
O      CPU_Input3:I0.3
ALD
A      T101
LPS
AR>    VD86, 0.1
EU
MOVW   +10, VW174
MOVR   VD86, VD108
S      M3.1, 1
LPP
AR=    VD86, 0.0
S      M2.1, 1
Network 37
LD     T102
EU
MOVR   VD104, VD404
R      M3.0, 1
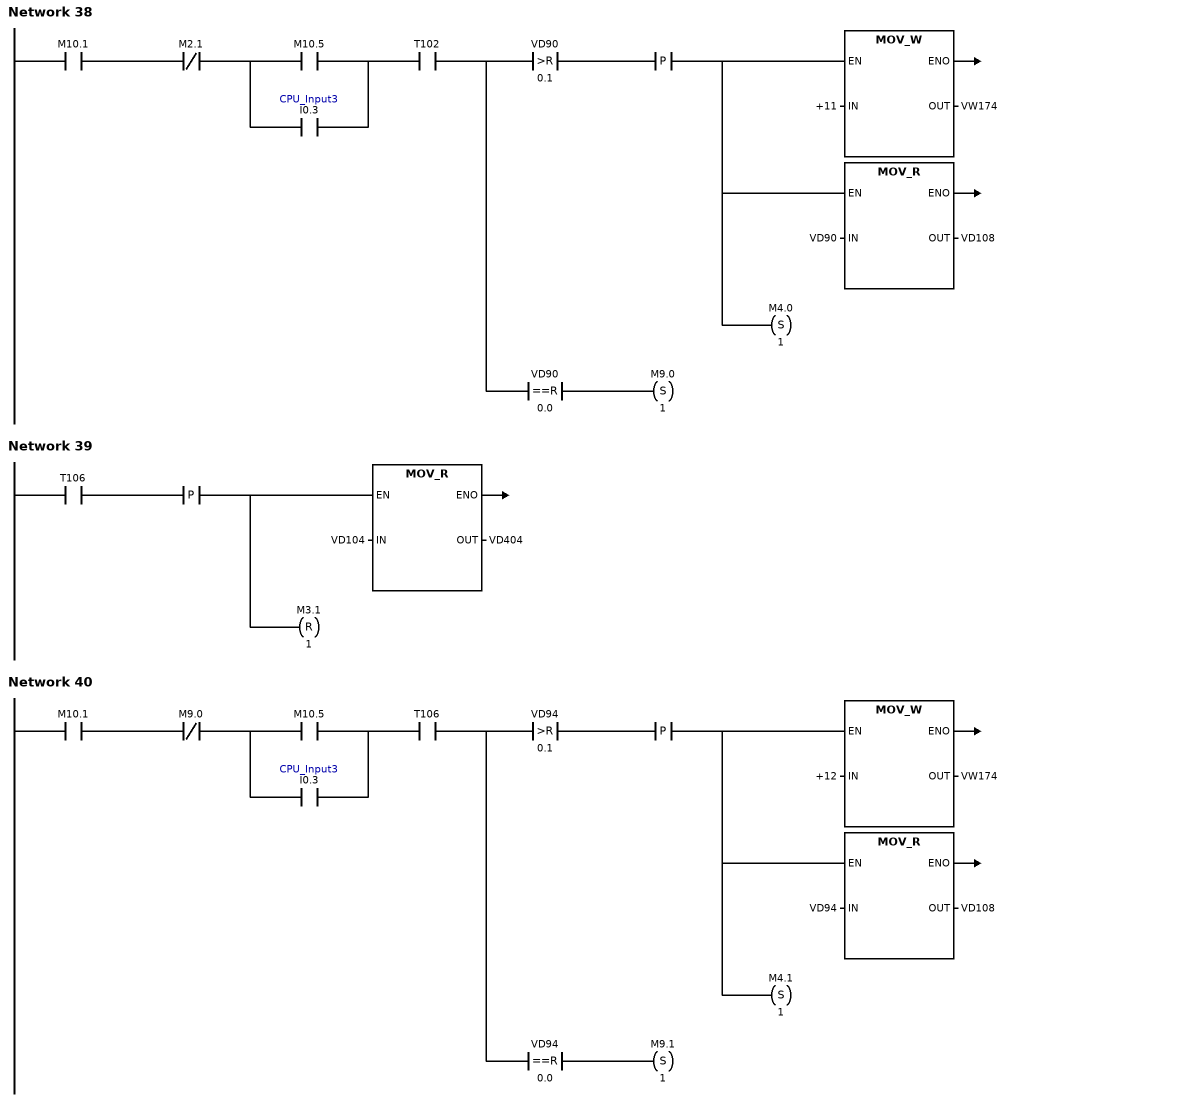
Network 38
LD     M10.1
AN     M2.1
LD     M10.5
O      CPU_Input3:I0.3
ALD
A      T102
LPS
AR>    VD90, 0.1
EU
MOVW   +11, VW174
MOVR   VD90, VD108
S      M4.0, 1
LPP
AR=    VD90, 0.0
S      M9.0, 1
Network 39
LD     T106
EU
MOVR   VD104, VD404
R      M3.1, 1
Network 40
LD     M10.1
AN     M9.0
LD     M10.5
O      CPU_Input3:I0.3
ALD
A      T106
LPS
AR>    VD94, 0.1
EU
MOVW   +12, VW174
MOVR   VD94, VD108
S      M4.1, 1
LPP
AR=    VD94, 0.0
S      M9.1, 1
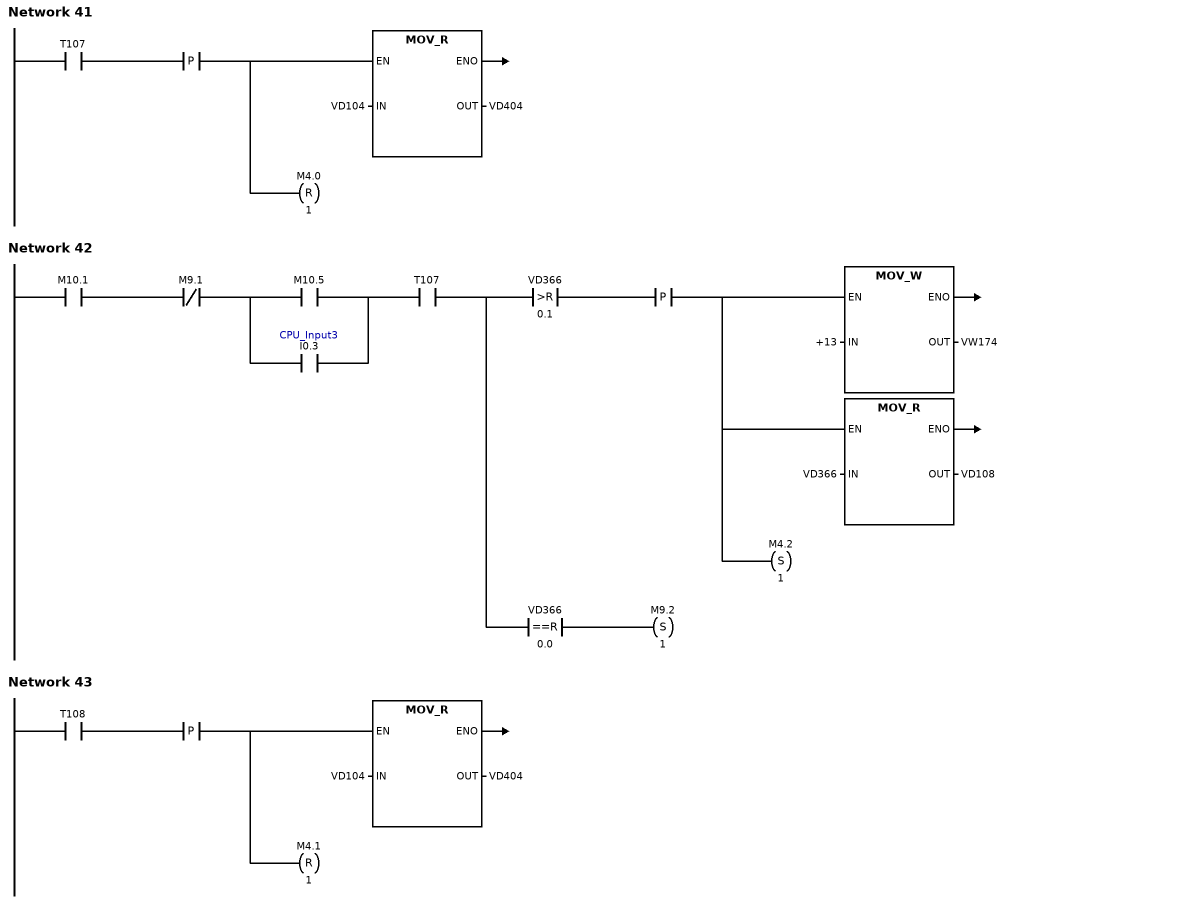
Network 41
LD     T107
EU
MOVR   VD104, VD404
R      M4.0, 1
Network 42
LD     M10.1
AN     M9.1
LD     M10.5
O      CPU_Input3:I0.3
ALD
A      T107
LPS
AR>    VD366, 0.1
EU
MOVW   +13, VW174
MOVR   VD366, VD108
S      M4.2, 1
LPP
AR=    VD366, 0.0
S      M9.2, 1
Network 43
LD     T108
EU
MOVR   VD104, VD404
R      M4.1, 1
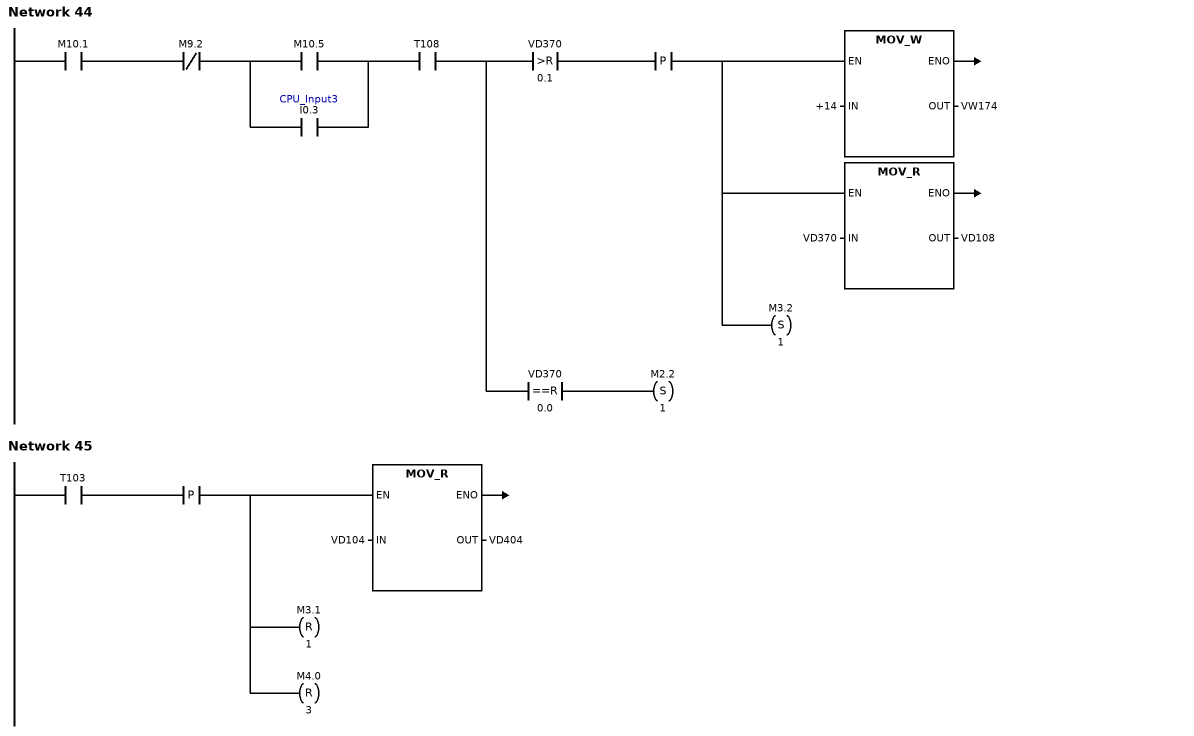
Network 44
LD     M10.1
AN     M9.2
LD     M10.5
O      CPU_Input3:I0.3
ALD
A      T108
LPS
AR>    VD370, 0.1
EU
MOVW   +14, VW174
MOVR   VD370, VD108
S      M3.2, 1
LPP
AR=    VD370, 0.0
S      M2.2, 1
Network 45
LD     T103
EU
MOVR   VD104, VD404
R      M3.1, 1
R      M4.0, 3
